// Mitsubishi GX Works2 project: TH06   PLC: FX2N/FX2NC

PROGRAM MAIN
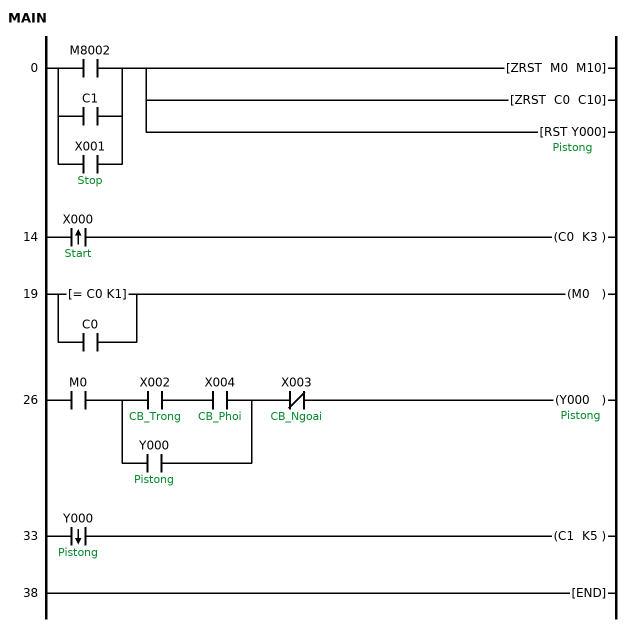
0     LD      M8002
      OR      C1
      OR      X001  ; Stop
      ZRST    M0 M10
      ZRST    C0 C10
      RST     Y000  ; Pistong
14    LDP     X000  ; Start
      OUT     C0 K3
19    LD=     C0 K1
      OR      C0
      OUT     M0
26    LD      M0
      LD      X002  ; CB_Trong
      AND     X004  ; CB_Phoi
      OR      Y000  ; Pistong
      ANB
      ANI     X003  ; CB_Ngoai
      OUT     Y000  ; Pistong
33    LDF     Y000  ; Pistong
      OUT     C1 K5
38    END
END_PROGRAM
